TYPE ST_StationReturn :
STRUCT
	Done	: BOOL;
	stState	: INT;
END_STRUCT
END_TYPE

(* stored: Version 1.1.0.1
   DUT ST_StationReturn: Id {15e1eb12-7a20-4052-b551-014221c39a0e} *)
